{attribute 'hide_all_locals'}
FUNCTION_BLOCK LINAXIS_JSC_XENAX EXTENDS FB_3_ROB_AXIS_LIN
VAR_INPUT
    SETTINGS : stSettings_LinAxis := (
        LinearStandStillLimit := 1.0,
        SafePositionTolerance := 1.0,
        StandardUnits := (
            Position := eUnit.mm,
            Orientation := eUnit.rad,
            Joint := eUnit.mm,
            LinearVelocity := eUnit.mm,
            AngularVelocity := eUnit.rad,
            JointVelocity := eUnit.mm,
            LinearAcceleration := eUnit.mm,
            AngularAcceleration := eUnit.rad,
            JointAcceleration := eUnit.mm));
    ReferenceMode : INT := gcJS_MC.jsmcREFERENCE_MODE_DONT_CHANGE;
    PowerOverride : LREAL := 100.0;
END_VAR
VAR_OUTPUT
    AXIS_COMM : FB_3_COMM_AXIS_JSC_XENAX;
END_VAR

VAR
	NCAxis: AXIS_REF;
END_VAR



AXIS_COMM(
    ReferenceMode := ReferenceMode,
    PowerOverride := PowerOverride,
    StopVelocityTolerance := SETTINGS.LinearStandStillLimit);
COMM := ADR(AXIS_COMM);
SET_A := SETTINGS;
_pSettingsLinAxis := ADR(SETTINGS);

Powered := AXIS_COMM.Powered;
Homed := AXIS_COMM.Homed;
ActualAxisPosition := AXIS_COMM.ActualPosition;
_axisActualVelocity := AXIS_COMM.ActualVelocity;

CYCLIC_LIN_AXIS();

METHOD CommandHandler : UINT
VAR_INPUT
    Cmd : eCommands;
    Settings : stCommand_Settings;
END_VAR
VAR
    NewCommandID : UINT;
    TargetPosition : LREAL;
    TargetValid : BOOL;
    EffectiveVelocity : LREAL;
    EffectiveAcceleration : LREAL;
    Accepted : BOOL;
END_VAR
CommandHandler := 0;
IF NOT PrepareAxisCommand(
    Cmd := Cmd,
    Settings := Settings,
    NewCommandID => NewCommandID,
    TargetPosition => TargetPosition,
    TargetValid => TargetValid,
    EffectiveVelocity => EffectiveVelocity,
    EffectiveAcceleration => EffectiveAcceleration) THEN RETURN; END_IF

CASE Cmd OF
    eCommands.MoveL, eCommands.MoveJ, eCommands.MoveJJoints:
        Accepted := AXIS_COMM.SendMoveAbsolute(
            CommandID := NewCommandID,
            Position := TargetPosition,
            Velocity := EffectiveVelocity,
            Acceleration := EffectiveAcceleration,
            Deceleration := SET_A.DefaultDeceleration,
            Jerk := SET_A.DefaultJerk);
    eCommands.MoveLRelativ, eCommands.MoveJRelativ:
        Accepted := AXIS_COMM.SendMoveRelative(
            CommandID := NewCommandID,
            Distance := Settings.Pose.x,
            Velocity := EffectiveVelocity,
            Acceleration := EffectiveAcceleration,
            Deceleration := SET_A.DefaultDeceleration,
            Jerk := SET_A.DefaultJerk);
    eCommands.Homing:
        Accepted := AXIS_COMM.SendHome(CommandID := NewCommandID);
END_CASE

IF Accepted THEN
    CommandHandler := CommitAxisCommand(
        NewCommandID := NewCommandID,
        TargetPosition := TargetPosition,
        TargetValid := TargetValid);
END_IF
END_METHOD

METHOD PROTECTED OnActivate : eResult
VAR
    eParentResult : eResult;
    myResult : eResult;
END_VAR


eParentResult := SUPER^.OnActivate();
myResult := eResult.NONE;

IF eParentResult <> eResult.SUCCESS THEN
    OnActivate := eParentResult;
    RETURN;
END_IF

AXIS_COMM.Power(Enable := FALSE);
IF NOT AXIS_COMM.Powered THEN
    myResult := eResult.SUCCESS;
END_IF

OnActivate := CombineResults(eParentResult, myResult);
END_METHOD

METHOD PROTECTED OnConfigure : eResult
VAR
    eParentResult : eResult;
    myResult : eResult;
END_VAR


eParentResult := SUPER^.OnConfigure();

IF NOT ValidateConfiguration() THEN
    myResult := eResult.FAILURE;
ELSE
    myResult := eResult.SUCCESS;
END_IF

OnConfigure := CombineResults(eParentResult, myResult);
END_METHOD

METHOD PROTECTED OnDeactivate : eResult
VAR
    eParentResult : eResult;
    myResult : eResult;
END_VAR
eParentResult := SUPER^.OnDeactivate();
myResult := eResult.NONE;

IF (ABS(AXIS_COMM.ActualVelocity) > SETTINGS.LinearStandStillLimit) OR AXIS_COMM.Busy THEN
    AXIS_COMM.StopMotion();
ELSE
    AXIS_COMM.Power(Enable := FALSE);
    IF NOT AXIS_COMM.Powered THEN
        myResult := eResult.SUCCESS;
    END_IF
END_IF

OnDeactivate := CombineResults(eParentResult, myResult);
END_METHOD

METHOD PROTECTED OnError : eResult
VAR
    eParentResult : eResult;
    myResult : eResult;
END_VAR
eParentResult := SUPER^.OnError();
myResult := eResult.NONE;

IF eParentResult <> eResult.SUCCESS THEN
    OnError := eParentResult;
    RETURN;
END_IF

IF AXIS_COMM.MESSENGER.HasActivError THEN
    AXIS_COMM.ResetAxis();
    myResult := eResult.NONE;
ELSE
    myResult := eResult.SUCCESS;
END_IF

OnError := CombineResults(eParentResult, myResult);
END_METHOD

END_FUNCTION_BLOCK

(* stored: Version 1.1.0.1, ProductVersion 3.1.4026.18
   POU LINAXIS_JSC_XENAX: Id {712fd3e6-7338-4ca3-919d-2d810e67e743}, SpecialFunc None
   Folder StateControl: Id {6131d21d-c55f-45df-8830-28d32c904ab8}
   Method CommandHandler: Id {50cb4440-da35-435c-af47-e6ce802d0dfd}
   Method OnActivate: Id {d3390fde-8c30-4f7b-b731-26ae87a488dd}
   Method OnConfigure: Id {58e8f349-71d5-46a4-8fb8-1145251f6bc0}
   Method OnDeactivate: Id {3e44d03e-f4bc-4817-b277-9318a9642557}
   Method OnError: Id {3b385f77-c2da-49d6-b0ac-25dcdd06a303} *)
